(*udt (user defined type) for all generic EOAT (End of Arm Tools)
	auth. Brent Lekx-Toniolo of Sodecia GTAC

------------------------------------------------------------------------
REVISION NOTES:

	Version 20151103:
	- initial concept, b.lekx-toniolo	
	Version 20170607
	- unknown changes or editor
------------------------------------------------------------------------

*)

TYPE udt_EOATxx_Image_20170607 :
	STRUCT
			(*Input nodes*)
			N01: udt_EP1008_002_v2;
			N02: udt_EP1008_002_v2;
			N03: udt_EP1008_002_v2;
			N04: udt_EP1008_002_v2;
			N05: udt_EP1008_002_v2;
			N06: udt_EP1008_002_v2;
			N07: udt_EP1008_002_v2;
			N08: udt_EP1008_002_v2;
			N09: udt_EP1008_002_v2;

			(*Valve Bank*)
			N100: udt_SMC_EX260_ValveBank;
			N100_STAT: udt_SMC_EX260_STAT;
			(*Cable Break States*)
			ECatSlave_Cable_Breaks: ARRAY[0..1] OF DINT;
			(*Node Counts*)
			NodeLayout:udt_ECATNodeData_20221507;
			NodeState:ARRAY[0..63] OF UINT;
			Input_Node_Count: UDINT;
			Safety_Node_Count:Udint;
			VB_Node_Count: UDINT;

			
			(*Developed Data*)
			CLFaults1: UDINT;
			CLFaults2: UDINT;
			CLFaults3: UDINT;
			CLFaults4: UDINT;
			CLFaulted: UDINT;
			PPFaults: UDINT;
			PPFaulted: UDINT;
			(*ID*)
			ID: UINT;
			strID: STRING[255];

	END_STRUCT
END_TYPE

(* stored: Version 1.1.0.1, ProductVersion 3.1.4024.9
   DUT udt_EOATxx_Image_20170607: Id {b7ccb285-ff27-44cd-8719-7628726e919b} *)
